{attribute addProperty BoxType "EL1918-0000-0016"}
{attribute addProperty Id "FSoE_CommandUSINT811FSIN_Module_1_InputBIT10.1251FSIN_Module_1_Module_FaultBIT10.1251FSIN_Module_2_InputBIT10.1251FSIN_Module_2_Module_FaultBIT10.1251FSIN_Module_3_InputBIT10.1251FSIN_Module_3_Module_FaultBIT10.1251FSIN_Module_4_InputBIT10.1251FSIN_Module_4_Module_FaultBIT10.1251FSIN_Module_5_InputBIT10.1251FSIN_Module_5_Module_FaultBIT10.1251FSIN_Module_6_InputBIT10.1251FSIN_Module_6_Module_FaultBIT10.1251FSIN_Module_7_InputBIT10.1251FSIN_Module_7_Module_FaultBIT10.1251FSIN_Module_8_InputBIT10.1251FSIN_Module_8_Module_FaultBIT10.1251FSoE_CRC_000UINT1623FSoE_Connection_IDUINT1622"}
{attribute addProperty CRC "73487565"}
{attribute addProperty SizeInBites "56"}
{attribute addProperty SizeInBytes "7"}
TYPE FSOE_046154CD :
STRUCT
	{attribute addProperty Name "FSoE_Command"}
	FSoE_Command : USINT;
	{attribute addProperty Name "FSIN_Module_1_Input"}
	FSIN_Module_1_Input : BIT;
	{attribute addProperty Name "FSIN_Module_1_Module_Fault"}
	FSIN_Module_1_Module_Fault : BIT;
	{attribute addProperty Name "FSIN_Module_2_Input"}
	FSIN_Module_2_Input : BIT;
	{attribute addProperty Name "FSIN_Module_2_Module_Fault"}
	FSIN_Module_2_Module_Fault : BIT;
	{attribute addProperty Name "FSIN_Module_3_Input"}
	FSIN_Module_3_Input : BIT;
	{attribute addProperty Name "FSIN_Module_3_Module_Fault"}
	FSIN_Module_3_Module_Fault : BIT;
	{attribute addProperty Name "FSIN_Module_4_Input"}
	FSIN_Module_4_Input : BIT;
	{attribute addProperty Name "FSIN_Module_4_Module_Fault"}
	FSIN_Module_4_Module_Fault : BIT;
	{attribute addProperty Name "FSIN_Module_5_Input"}
	FSIN_Module_5_Input : BIT;
	{attribute addProperty Name "FSIN_Module_5_Module_Fault"}
	FSIN_Module_5_Module_Fault : BIT;
	{attribute addProperty Name "FSIN_Module_6_Input"}
	FSIN_Module_6_Input : BIT;
	{attribute addProperty Name "FSIN_Module_6_Module_Fault"}
	FSIN_Module_6_Module_Fault : BIT;
	{attribute addProperty Name "FSIN_Module_7_Input"}
	FSIN_Module_7_Input : BIT;
	{attribute addProperty Name "FSIN_Module_7_Module_Fault"}
	FSIN_Module_7_Module_Fault : BIT;
	{attribute addProperty Name "FSIN_Module_8_Input"}
	FSIN_Module_8_Input : BIT;
	{attribute addProperty Name "FSIN_Module_8_Module_Fault"}
	FSIN_Module_8_Module_Fault : BIT;
	{attribute addProperty Name "FSoE_CRC_000"}
	FSoE_CRC_000 : UINT;
	{attribute addProperty Name "FSoE_Connection_ID"}
	FSoE_Connection_ID : UINT;
END_STRUCT
END_TYPE

(* stored: Version 1.2.0.0, ProductVersion 3.1.4024.9
   DUT FSOE_046154CD: Id {e0478f08-c8ab-420f-8cb9-2e93010a63f6} *)
